(* compensation not necessarily finished if axis stops (new modes available) - 2009-08-13 KSt *)
(*	IF NOT F_AxisHasJob(Axis.NcToPlc.StateDWord) THEN
		/* command aborted, move has been stopped before superposition finished (KSt, 12.01.2004) */
		CommandAborted := TRUE;
		iState := STATE_INITIALIZATION;
	END_IF
*)

STATE_WAITING : (* 2009-10-06 KSt  - state added for axes coupled to actual position (encoder axes or disabled axes) *)
	(* decide if superposition was completed or aborted in case of axes coupled to actual position (encoder axes or disabled axes) *)
	IF NOT F_AxisIsMoving(Axis.NcToPlc.StateDWord) THEN (* 2009-10-06 KSt *)
		(* command aborted, motion ended before superposition was finished because the axis is not moving any longer *)
		CommandAborted := TRUE;
	ELSE
		(* the initial HasJob or Moving state was the same as at end of compensation - assume that superposition completed *)
		Done := TRUE;
	END_IF
	CompensationStarted := FALSE;
	iState := STATE_INITIALIZATION;

ELSE  (* CASE : Unknown program state *)
	Error := TRUE;
	ErrorID := 16#FFFFFFFF;
	iState:= STATE_INITIALIZATION;
END_CASE

ADSbusy := fbAdsReadWrite.BUSY;
IF iState=STATE_INITIALIZATION THEN
	(* reset Busy immediately  when sequence ends *)
	IF Busy THEN
		LastExecutionResult.Done := Done;
		LastExecutionResult.CommandAborted := CommandAborted;
		LastExecutionResult.Error := Error;
		LastExecutionResult.ErrorID := ErrorID;
	END_IF
	Busy := FALSE;
	Active := FALSE;
END_IF
END_FUNCTION_BLOCK

(* POU MC_OverrideFilter, ST *)
FUNCTION_BLOCK MC_OverrideFilter
VAR_INPUT
	(* variables *)
	OverrideValueRaw		: DINT;
	(* parameter *)
	LowerOverrideThreshold	: DINT	:= 0;			(* 0...32767 digits *)
	UpperOverrideThreshold	: DINT	:= 32767;		(* 0...32767 digits *)
	OverrideSteps			: UDINT	:= 200;		(* 200 steps => 0.5 percent *)
	OverrideRecoveryTime	: TIME	:= T#150ms;	(* 150 ms *)
END_VAR
VAR_OUTPUT
	OverrideValueFiltered		: DWORD;			(* 0...1000000 counts *)
	OverridePercentFiltered	: LREAL;				(* 0...100 % *)
	Error					: BOOL;
	ErrorID					: UDINT;
END_VAR
VAR
	bFirstCycle				: BOOL := TRUE;
	bThresholdActive			: BOOL := TRUE;
	InternalOverrideValueRaw	: DINT;
	LastOverrideValueRaw		: DINT := 16#FFFF;
	OverrideRange			: DINT;
END_VAR
{library private}
VAR
	fbTimer					: TON;
END_VAR
(* default value *)
Error	:= FALSE;
ErrorID	:= MC_ERROR_NO_ERROR;

(* check parameter / error handling:   'UpperOverrideThreshold > LowerOverrideThreshold'  AND  'OverrideSteps > 1'  *)
IF( (LowerOverrideThreshold >= UpperOverrideThreshold) OR (OverrideSteps <= 1) )THEN
	OverrideValueFiltered		:= 0;
	OverridePercentFiltered	:= 0.0;
	Error	:= TRUE;
	ErrorID	:= MC_ERROR_PARAMETER_NOT_CORRECT;
	RETURN;
END_IF;

(* first cycle: timer must be elapsed *)
IF ( bFirstCycle ) THEN
	fbTimer( IN:=TRUE, PT:= T#0s );
	bFirstCycle := FALSE;
END_IF;

IF ( OverrideValueRaw >= UpperOverrideThreshold ) THEN
	InternalOverrideValueRaw := UpperOverrideThreshold;
	bThresholdActive := TRUE;
ELSIF ( OverrideValueRaw <= LowerOverrideThreshold ) THEN
	InternalOverrideValueRaw := LowerOverrideThreshold;
	bThresholdActive := TRUE;
ELSE
	InternalOverrideValueRaw := OverrideValueRaw;
	bThresholdActive := FALSE;
END_IF;

fbTimer( IN:=TRUE, PT:= OverrideRecoveryTime );
IF( fbTimer.Q = TRUE OR bThresholdActive )THEN
	OverrideRange := UpperOverrideThreshold - LowerOverrideThreshold;
(*	IF (  bThresholdActive OR ABS( InternalRawOverrideValue - LastRawOverrideValue ) >= (0.5 * OverrideRange / OverrideSteps)  ) THEN *)
	IF (  bThresholdActive OR ABS( InternalOverrideValueRaw - LastOverrideValueRaw ) >= ( OverrideRange / OverrideSteps)  ) THEN
		OverrideValueFiltered := ((InternalOverrideValueRaw - LowerOverrideThreshold) * 1000 / OverrideRange) * 1000;
		OverridePercentFiltered := DWORD_TO_LREAL( OverrideValueFiltered ) * 0.0001;
		LastOverrideValueRaw := InternalOverrideValueRaw;
		fbTimer( IN:=FALSE, PT:= OverrideRecoveryTime );
	END_IF;
END_IF;
END_FUNCTION_BLOCK

(* POU MC_Power, ST *)
FUNCTION_BLOCK MC_Power
(*
	Function block defined by PLCopen Part 1 - Function blocks for motion control

	This Function Block controls the power stage (on or off).
*)
VAR_IN_OUT
	Axis				:	AXIS_REF;	(* B *)
END_VAR
VAR_INPUT
	Enable			:	BOOL;	(* B *)
	Enable_Positive	:	BOOL;	(* E *)
	Enable_Negative	:	BOOL;	(* E *)
	Override			:	LREAL	(* V *) 	:= 100.0; (* in percent - Beckhoff proprietary input *)
	BufferMode		:	MC_BufferMode;	(* E *)
END_VAR
VAR_OUTPUT
	Status			:	BOOL;	(* B *)
	Busy			: 	BOOL;	(* E *)
	Active			: 	BOOL;	(* E *)
	Error			:	BOOL;	(* B *)
	ErrorID			:	UDINT;	(* E *)
END_VAR
{library private}
VAR
	EnableTimeout: TON;
	EnableOffOnDelay: TP;
	iOverride: DINT;
END_VAR
(*EnableTimeout(IN:=Enable, PT:=T#10s);*)	(* timout if axis doesn't get ready after Enable *)
EnableTimeout(IN:=Enable AND NOT Status AND Axis.NcToPlc.CoupleState=0, PT:=T#10s);	(* timout if axis doesn't get ready after Enable - just for single axes - KSt 2010-03-11 *)
EnableOffOnDelay(IN:= NOT Enable );	(* minimum delay between disable end re-Enable -  don't initialize before first enable *)

IF Enable THEN
	Busy := TRUE;
	Status := FALSE;
	ErrorID := 0;
	Error := FALSE;
	EnableOffOnDelay.PT:=T#50ms;	(* initialize not before first enable *)

	(* set override *)
	iOverride := LREAL_TO_UDINT(Override*10000);
	(* double check override with real and integer number because conversion may fail *)
	IF (Override < -1) OR (Override > 101) THEN	(* check real number with tolerance *)
		ErrorID := MC_ERROR_PARAMETER_NOT_CORRECT;
		Error := TRUE;
	ELSIF (iOverride < 0) OR (iOverride > 1000000) THEN	(* check integer number without tolerance *)
		ErrorID := MC_ERROR_PARAMETER_NOT_CORRECT;
		Error := TRUE;
	ELSE
		Axis.PlcToNc.Override := iOverride;
	END_IF;

	(* set enabling flags *)
	Axis.PlcToNc.ControlDWord.0 := Enable;
	Axis.PlcToNc.ControlDWord.1 := Enable_Positive;
	Axis.PlcToNc.ControlDWord.2 := Enable_Negative;

	(* set status bit *)
	(* IF  F_AxisIsReady(StateDWord := Axis.NcToPlc.StateDWord) THEN *) (* Axis ready*) 	(* 2008-12-18 KSt *)
	IF  F_AxisControlLoopClosed(StateDWord := Axis.NcToPlc.StateDWord) THEN (* Axis ready*) 	(* 2008-12-18 KSt *)
		(* status is TRUE if no error and a minimum of EnableOffOnDelay.PT (50 ms) after last recent disable *)
		Status := NOT Error AND NOT EnableOffOnDelay.Q; (* exclusive outputs *)
	ELSIF Axis.Status.ErrorID <> 0 THEN (* 2009-01-29 KSt *)
		Status := FALSE;
		Error := TRUE;
		ErrorID := Axis.Status.ErrorID;
	ELSIF EnableTimeout.Q THEN
		(* timeout after enable *)
		Status := FALSE;
		Error := TRUE;
		ErrorID := MC_ERROR_AXIS_IS_NOT_READY;
	END_IF;

ELSE (* NOT Enable *)
	(* if BufferMode=Buffered wait for current command beeing finished *)
	IF BufferMode = MC_Aborting OR NOT F_AxisHasJob(Axis.NcToPlc.StateDWord) THEN
		Axis.PlcToNc.ControlDWord:= CLEARBIT32(Axis.PlcToNc.ControlDWord,0);
		Axis.PlcToNc.ControlDWord:= CLEARBIT32(Axis.PlcToNc.ControlDWord,1);
		Axis.PlcToNc.ControlDWord:= CLEARBIT32(Axis.PlcToNc.ControlDWord,2);
		(* Override  0 % *)
		Axis.PlcToNc.Override := 0;
		Status := FALSE;
		Busy := FALSE;
		Error := FALSE;			(* reset at falling edge of Execute *)
		ErrorID := 0;
	END_IF
END_IF;

Active:=TRUE;
END_FUNCTION_BLOCK

(* POU MC_PowerStepper, ST *)
FUNCTION_BLOCK MC_PowerStepper
VAR_IN_OUT
	Axis		:	AXIS_REF;
END_VAR
VAR_INPUT
	Enable			:	BOOL;
	Enable_Positive	:	BOOL;
	Enable_Negative	:	BOOL;
	Override			:	LREAL := 100.0; (* in percent *)
	DestallParams	:	ST_PowerStepperStruct;
	KL_Status		:	USINT;
	KL_Status2		:	UINT;
END_VAR
VAR_OUTPUT
	Status			:	BOOL;
	Error			:	BOOL;
	ErrorID			:	UDINT;
	Stalled			:	BOOL;
	StallError			:	BOOL;
END_VAR
VAR
	fbPower			:	MC_Power;
	ErrorCode		:	DWORD;
	fbWriteErrCode	:	ADSWRITE;
	nRefState		:	DWORD;
	fbWriteNonRef	:	ADSWRITE;
	fbReadParams	:	ADSREAD;
	fbWriteInstOvr		:	ADSWRITE;
	bAdsInitDone		:	BOOL;

	bOverTemp		:	BOOL;
	rtOverTemp		:	R_TRIG;
	bUnderVoltage	:	BOOL;
	rtUnderVoltage	:	R_TRIG;
	bOpenLoopA		:	BOOL;
	rtOpenLoopA		:	R_TRIG;
	bOpenLoopB		:	BOOL;
	rtOpenLoopB		:	R_TRIG;
	bOverCurrentA	:	BOOL;
	rtOverCurrentA	:	R_TRIG;
	bOverCurrentB	:	BOOL;
	rtOverCurrentB	:	R_TRIG;
	rtStallError		:	R_TRIG;
	bOldState		:	BOOL;

	bLagFilterInit		: 	BOOL;
	tonLagFilter		:	TON;
	tonNoLagFilter	:	TON;

	wState2			:	WORD;
	nAngle			:	INT;
	nOldAngle		:	INT;
	AngleDiff			:	INT;
	bInErrorState		:	BOOL;

	nParamIdx		:	INT;
	bParamEnabled	:	BOOL;
	fLagLimit			:	LREAL;
	fLagFilter			:	LREAL;
	nTries			:	INT;
	tTimeOut			:	TON;
END_VAR
(*
	Aufruf des Standard-Bausteins
*)
fbPower(
	Enable:=Enable,
	Enable_Positive:=Enable_Positive,
	Enable_Negative:=Enable_Negative,
	Override:=Override,
	Axis:=Axis);

(*
	Ein paar Vorbereitungen ...
*)
wState2:=UINT_TO_WORD(KL_Status2);
bInErrorState:=Axis.NcToPlc.ErrorCode<>0;
nAngle:=SHR(USINT_TO_BYTE(KL_Status),1) AND 7;
AngleDiff:=nAngle-nOldAngle;
nOldAngle:=nAngle;
IF((Axis.NcToPlc.StateDWord AND 16#0000001C)=16#0000001C)THEN		(* Ziel erreicht *)
	nTries:=0;
END_IF
IF((Axis.NcToPlc.StateDWord AND 16#00000080)=16#00000080)THEN		(* Stop *)
	nTries:=0;
END_IF

(* ======================================
	Parameter-Lademaschine
====================================== *)
IF(NOT Enable)THEN
	(*
		Reinitialisieren
	*)
	nParamIdx:=0;
	bParamEnabled:=FALSE;
	fbReadParams(
		NETID:='', PORT:=AMSPORT_R0_NCSAF, IDXGRP:=0, IDXOFFS:=0,
		LEN:=0, DESTADDR:=0,
		READ:=FALSE, TMOUT:=T#5s);
ELSE
	IF(NOT bParamEnabled)THEN
		CASE nParamIdx OF
			0:
				IF(NOT fbReadParams.READ)THEN
					fbReadParams.LEN:=SIZEOF(fLagLimit);
					fbReadParams.DESTADDR:=ADR(fLagLimit);
					fbReadParams.IDXGRP:=16#00004000+Axis.NcToPlc.AxisId;
					fbReadParams.IDXOFFS:=16#00020012;
					fbReadParams.READ:=TRUE;
				ELSIF(NOT fbReadParams.BUSY)THEN
					IF(fbReadParams.ERR)THEN
						fLagLimit:=5.0;
					END_IF
					fbReadParams.READ:=FALSE;
					nParamIdx:=nParamIdx+1;
				END_IF
				fbReadParams(NETID:='', PORT:=AMSPORT_R0_NCSAF, TMOUT:=T#5s);
			1:
				IF(NOT fbReadParams.READ)THEN
					fbReadParams.LEN:=SIZEOF(fLagFilter);
					fbReadParams.DESTADDR:=ADR(fLagFilter);
					fbReadParams.IDXGRP:=16#00004000+Axis.NcToPlc.AxisId;
					fbReadParams.IDXOFFS:=16#00020013;
					fbReadParams.READ:=TRUE;
				ELSIF(NOT fbReadParams.BUSY)THEN
					IF(fbReadParams.ERR)THEN
						fLagFilter:=0.1;
					END_IF
					fbReadParams.READ:=FALSE;
					nParamIdx:=nParamIdx+1;
					tonLagFilter(IN:=FALSE, PT:=T#10ms);
					tonNoLagFilter(IN:=NOT tonLagFilter.IN, PT:=T#10ms);
				END_IF
				fbReadParams(NETID:='', PORT:=AMSPORT_R0_NCSAF, TMOUT:=T#5s);
			ELSE
				bParamEnabled:=TRUE;
		END_CASE
	END_IF
END_IF

IF(fbPower.Error)THEN
	ErrorID := fbPower.ErrorID;
	Error := TRUE;
	Status := bAdsInitDone := FALSE;
ELSIF(NOT Enable)THEN
	ErrorID := 0;
	Error := Status := bAdsInitDone := FALSE;
ELSE
	(*
		Sicherstellen, dass die ADS-FBs initialisiert sind
	*)
	IF(NOT bAdsInitDone)THEN
		bAdsInitDone := TRUE;
		fbWriteNonRef(
			WRITE:=FALSE,
			NETID:='',
			PORT:=AMSPORT_R0_NCSAF,
			IDXGRP:=16#00004200+Axis.NcToPlc.AxisId,
			IDXOFFS:=16#0000001B,
			LEN:=SIZEOF(nRefState),
			SRCADDR:=ADR(nRefState),
			TMOUT:=T#5s,
			);
		fbWriteInstOvr(
			WRITE:=FALSE,
			NETID:='',
			PORT:=AMSPORT_R0_NCSAF,
			IDXGRP:=16#00004200+Axis.NcToPlc.AxisId,
			IDXOFFS:=16#00000029,
			LEN:=0,
			SRCADDR:=0,
			TMOUT:=T#5s,
			);
		fbWriteErrCode(
			WRITE:=FALSE,
			NETID:='',
			PORT:=AMSPORT_R0_NCSAF,
			IDXGRP:=16#00004200+Axis.NcToPlc.AxisId,
			IDXOFFS:=16#00000019,
			LEN:=SIZEOF(ErrorCode),
			SRCADDR:=ADR(ErrorCode),
			TMOUT:=T#5s,
			);
	END_IF

	(*
		Zentrales Versenden für Kommandos zur instantanen Override-Änderung
		Dies muss vor der Stelle des Test liegen, damit der Override-Wert im Mapping sicher angekommen ist,
		wenn dieses Kommando per ADS eintrifft.
	*)
	fbWriteInstOvr(
		NETID:='',
		PORT:=AMSPORT_R0_NCSAF,
		IDXGRP:=16#00004200+Axis.NcToPlc.AxisId,
		IDXOFFS:=16#00000029,
		LEN:=0,
		SRCADDR:=0,
		TMOUT:=T#5s,
		);
	IF(NOT fbWriteInstOvr.BUSY)THEN
		fbWriteInstOvr.WRITE:=FALSE;
	END_IF

	bLagFilterInit:=bLagFilterInit OR tonLagFilter.Q;

	IF(DestallParams.DestallEnable)THEN
		(*
			Stall Detection
		*)
		bOldState:=Stalled;
		CASE DestallParams.DestallDetectMode OF
			PwStDetectMode_Encoderless:
				Stalled:=ABS(AngleDiff)>=4;
			PwStDetectMode_Lagging:
				IF(bParamEnabled)THEN
					IF(fLagFilter<=0.001)THEN
						tonLagFilter(IN:=FALSE, PT:=T#10ms);
						tonNoLagFilter(IN:=NOT tonLagFilter.IN, PT:=T#10ms);
						Stalled:=ABS(Axis.NcToPlc.PosDiff)>=fLagLimit;
					ELSE
						tonLagFilter(IN:=(ABS(Axis.NcToPlc.PosDiff)>=fLagLimit), PT:=LREAL_TO_TIME(fLagFilter*1000.0));
						tonNoLagFilter(IN:=NOT tonLagFilter.IN, PT:=LREAL_TO_TIME(fLagFilter*1000.0));
						Stalled:=tonLagFilter.Q;
					END_IF
				ELSE
					tonLagFilter(IN:=FALSE, PT:=T#10ms);
					tonNoLagFilter(IN:=NOT tonLagFilter.IN, PT:=T#10ms);
					Stalled:=FALSE;
				END_IF
			ELSE
				Stalled:=FALSE;
		END_CASE
		IF(NOT bOldState AND Stalled)THEN
			nTries:=nTries+1;
		END_IF
		(*
			Stall Handling
		*)
		StallError:=StallError AND (bInErrorState  OR fbWriteErrCode.WRITE);
		bOldState:=StallError;
		CASE DestallParams.DestallMode OF
			PwStMode_None:
				StallError:=FALSE;
				tTimeOut(IN:=FALSE, PT:=T#10ms);
			PwStMode_SetError:
				StallError:=StallError OR Stalled;
				tTimeOut(IN:=FALSE, PT:=T#10ms);
			PwStMode_SetErrNonRef:
				StallError:=StallError OR Stalled;
				IF(Stalled AND ((Axis.NcToPlc.StateDWord AND 16#00000002)<>0) )THEN
					nRefState:=0;
					fbWriteNonRef.WRITE:=TRUE;
				END_IF
				tTimeOut(IN:=FALSE, PT:=T#10ms);
			PwStMode_UseOverride:
				IF(Stalled OR (bLagFilterInit AND NOT tonNoLagFilter.Q))THEN	(* HKP *)
					Axis.PlcToNc.Override := 0;
					fbWriteInstOvr.WRITE:=TRUE;
				END_IF
				tTimeOut(IN:=Stalled, PT:=MAX(DestallParams.Timeout, T#10ms));
				StallError:=StallError OR tTimeOut.Q;
				IF(nTries>DestallParams.Retries)THEN
					StallError:=TRUE;
				END_IF
		END_CASE

		IF(StallError AND NOT bOldState)THEN
			ADSLOGDINT((ADSLOG_MSGTYPE_ERROR OR ADSLOG_MSGTYPE_LOG), 'MC_PowerStepper (AxisID: %d) reporting error 0x4636 (stall error) !', Axis.NcToPlc.AxisId);
		END_IF
		rtStallError(CLK:=StallError AND NOT bInErrorState AND NOT fbWriteErrCode.WRITE);
		IF(rtStallError.Q)THEN
			ErrorCode:=16#00004636;
			fbWriteErrCode.WRITE:=TRUE;
		END_IF

	END_IF

	Status:=TRUE;
	IF(DestallParams.StatusMonEnable)THEN
		(*
			State Monitoring
		*)
		bOldState:=bOverTemp;
		bOverTemp:=(wState2 AND 2#0000000100000000)<>0;
		Status:=Status AND NOT bOverTemp;
		IF(bOverTemp AND NOT bOldState)THEN
			ADSLOGDINT((ADSLOG_MSGTYPE_ERROR OR ADSLOG_MSGTYPE_LOG), 'MC_PowerStepper (AxisID: %d) reporting error 0x4630 (overtemperature, KL terminal) !', Axis.NcToPlc.AxisId);
		END_IF
		rtOverTemp(CLK:=bOverTemp AND NOT bInErrorState AND NOT fbWriteErrCode.WRITE);
		IF(rtOverTemp.Q)THEN
			ErrorCode:=16#00004630;
			fbWriteErrCode.WRITE:=TRUE;
		END_IF
		bOverTemp:=bOverTemp AND (bInErrorState  OR fbWriteErrCode.WRITE);
		bOldState:=bUnderVoltage;
		bUnderVoltage:=(wState2 AND 2#0000001000000000)<>0;
		Status:=Status AND NOT bUnderVoltage;
		IF(bUnderVoltage AND NOT bOldState)THEN
						ADSLOGDINT((ADSLOG_MSGTYPE_ERROR OR ADSLOG_MSGTYPE_LOG), 'MC_PowerStepper (AxisID: %d) reporting error 0x4631 (bad supply voltage, KL terminal) !', Axis.NcToPlc.AxisId);
		END_IF
		rtUnderVoltage(CLK:=bUnderVoltage AND NOT bInErrorState AND NOT fbWriteErrCode.WRITE);
		IF(rtUnderVoltage.Q)THEN
			ErrorCode:=16#00004631;
			fbWriteErrCode.WRITE:=TRUE;
		END_IF
		bUnderVoltage:=bUnderVoltage AND (bInErrorState  OR fbWriteErrCode.WRITE);
		bOldState:=bOpenLoopA;
		bOpenLoopA:=(wState2 AND 2#0000010000000000)<>0;
		Status:=Status AND NOT bOpenLoopA;
		IF(bOpenLoopA AND NOT bOldState)THEN
			ADSLOGDINT((ADSLOG_MSGTYPE_ERROR OR ADSLOG_MSGTYPE_LOG), 'MC_PowerStepper (AxisID: %d) reporting error 0x4632 (open loop, phase A) !', Axis.NcToPlc.AxisId);
		END_IF
		rtOpenLoopA(CLK:=bOpenLoopA AND NOT bInErrorState AND NOT fbWriteErrCode.WRITE);
		IF(rtOpenLoopA.Q)THEN
			ErrorCode:=16#00004632;
			fbWriteErrCode.WRITE:=TRUE;
		END_IF
		bOpenLoopA:=bOpenLoopA AND (bInErrorState  OR fbWriteErrCode.WRITE);
		bOldState:=bOpenLoopB;
		bOpenLoopB:=(wState2 AND 2#0000100000000000)<>0;
		Status:=Status AND NOT bOpenLoopB;
		IF(bOpenLoopB AND NOT bOldState)THEN
			ADSLOGDINT((ADSLOG_MSGTYPE_ERROR OR ADSLOG_MSGTYPE_LOG), 'MC_PowerStepper (AxisID: %d) reporting error 0x4633 (open loop, phase B) !', Axis.NcToPlc.AxisId);
		END_IF
		rtOpenLoopB(CLK:=bOpenLoopB AND NOT bInErrorState AND NOT fbWriteErrCode.WRITE);
		IF(rtOpenLoopB.Q)THEN
			ErrorCode:=16#00004633;
			fbWriteErrCode.WRITE:=TRUE;
		END_IF
		bOpenLoopB:=bOpenLoopB AND (bInErrorState  OR fbWriteErrCode.WRITE);
		bOldState:=bOverCurrentA;
		bOverCurrentA:=(wState2 AND 2#0001000000000000)<>0;
		Status:=Status AND NOT bOverCurrentA;
		IF(bOverCurrentA AND NOT bOldState)THEN
			ADSLOGDINT((ADSLOG_MSGTYPE_ERROR OR ADSLOG_MSGTYPE_LOG), 'MC_PowerStepper (AxisID: %d) reporting error 0x4634 (overcurrent, phase A) !', Axis.NcToPlc.AxisId);
		END_IF
		rtOverCurrentA(CLK:=bOverCurrentA AND NOT bInErrorState AND NOT fbWriteErrCode.WRITE);
		IF(rtOverCurrentA.Q)THEN
			ErrorCode:=16#00004634;
			fbWriteErrCode.WRITE:=TRUE;
		END_IF
		bOverCurrentA:=bOverCurrentA AND (bInErrorState  OR fbWriteErrCode.WRITE);
		bOldState:=bOverCurrentB;
		bOverCurrentB:=(wState2 AND 2#0010000000000000)<>0;
		Status:=Status AND NOT bOverCurrentB;
		IF(bOverCurrentB AND NOT bOldState)THEN
			ADSLOGDINT((ADSLOG_MSGTYPE_ERROR OR ADSLOG_MSGTYPE_LOG), 'MC_PowerStepper (AxisID: %d) reporting error 0x4635 (overcurrent, phase B) !', Axis.NcToPlc.AxisId);
		END_IF
		rtOverCurrentB(CLK:=bOverCurrentB AND NOT bInErrorState AND NOT fbWriteErrCode.WRITE);
		IF(rtOverCurrentB.Q)THEN
			ErrorCode:=16#00004635;
			fbWriteErrCode.WRITE:=TRUE;
		END_IF
		bOverCurrentB:=bOverCurrentB AND (bInErrorState  OR fbWriteErrCode.WRITE);
	END_IF

	(*
		Zentrale Versendung von Achs-ErrorCodes
	*)
	fbWriteErrCode(
		NETID:='',
		PORT:=AMSPORT_R0_NCSAF,
		IDXGRP:=16#00004200+Axis.NcToPlc.AxisId,
		IDXOFFS:=16#00000019,
		LEN:=SIZEOF(ErrorCode),
		SRCADDR:=ADR(ErrorCode),
		TMOUT:=T#5s,
		);
	IF(bInErrorState)THEN
		fbWriteErrCode.WRITE:=FALSE;
	END_IF

	(*
		Zentrale Versendung von Referenz-Resets
	*)
	fbWriteNonRef(
		NETID:='',
		PORT:=AMSPORT_R0_NCSAF,
		IDXGRP:=16#00004200+Axis.NcToPlc.AxisId,
		IDXOFFS:=16#0000001B,
		LEN:=SIZEOF(nRefState),
		SRCADDR:=ADR(nRefState),
		TMOUT:=T#5s,
		);
	IF(NOT fbWriteNonRef.BUSY)THEN
		fbWriteNonRef.WRITE:=FALSE;
	END_IF

END_IF
END_FUNCTION_BLOCK

(* POU MC_ReadActualPosition, ST *)
FUNCTION_BLOCK MC_ReadActualPosition
(*	This Function Block returns the actual position. *)
VAR_IN_OUT
	Axis			:	AXIS_REF;	(* B *)
END_VAR
VAR_INPUT
	Enable		:	BOOL;		(* B *)
END_VAR
VAR_OUTPUT
	Valid		:	BOOL;		(* B *)
	Busy		:	BOOL;		(* E *)
	Error		:	BOOL;		(* B *)
	ErrorID		:	UDINT;		(* E *)
	Position		:	LREAL;		(* B *)
END_VAR
VAR
END_VAR
Error := FALSE;
ErrorID := 0;
IF Enable THEN
	Busy := TRUE;
	Position := Axis.NcToPlc.ActPos;
	Valid := TRUE;
ELSE
	Busy := FALSE;
	Position := 0.0;
	Valid := FALSE;
END_IF;
END_FUNCTION_BLOCK

(* POU MC_ReadActualVelocity, ST *)
FUNCTION_BLOCK MC_ReadActualVelocity
(*
	This Function Block returns the value of the actual velocity as long as Enable is 
	set. Valid is true when the data-output ActualVelocity is valid. If Enable is Reset, the 
	data loses its validity, and Valid is also reset, no matter if new data is available.
*)
VAR_IN_OUT
	Axis			:	AXIS_REF;	(* B *)
END_VAR
VAR_INPUT
	Enable 		: 	BOOL;	(* B *)
END_VAR
VAR_OUTPUT
	Valid 		: 	BOOL;	(* B *)
	Busy 		: 	BOOL;	(* E *)
	Error 		: 	BOOL;	(* B *)
	ErrorID 		: 	UDINT;	(* E *)
	ActualVelocity : 	LREAL;	(* B *)
END_VAR
VAR
END_VAR
Error := FALSE;
ErrorID := 0;
IF Enable THEN
	Busy := TRUE;
	Valid := TRUE;
	ActualVelocity := Axis.NcToPlc.ActVelo;
ELSE
	Busy := FALSE;
	Valid := FALSE;
	ActualVelocity := 0;
END_IF
END_FUNCTION_BLOCK

(* POU MC_ReadAxisComponents, ST *)
FUNCTION_BLOCK  MC_ReadAxisComponents
VAR_IN_OUT
	AxisComponents 	: 	ST_AxisComponents;
	Axis				:	AXIS_REF;
END_VAR
VAR_INPUT
	Execute: BOOL;
END_VAR
VAR_OUTPUT
	Done : BOOL;
	Busy: BOOL;
	Error : BOOL;
	ErrorID : UDINT;
END_VAR
VAR
	TriggerExecute: R_TRIG;
	state: _E_TcMC_STATES := STATE_INITIALIZATION;
	fbAdsRead		: 	ADSREAD;
END_VAR
TriggerExecute(CLK:=Execute);

CASE state OF
	STATE_INITIALIZATION:
		IF NOT Execute THEN
			Done := FALSE;
			Error := FALSE;	(* reset at falling edge of Execute *)
			ErrorID := 0;
		END_IF
		IF TriggerExecute.Q THEN
			Done := FALSE;
			Busy := TRUE;
			Error := FALSE;
			ErrorID := 0;
			fbAdsRead(READ:=FALSE);
		END_IF
		IF Busy THEN
			fbAdsRead(
				NETID:= TcMcGlobal.NCNETID_TCMC,
				PORT:= TcMcGlobal.NCPORT_TCMC,
				IDXGRP:=TcMcGlobal.Axis.Parameter.IDXGRP+Axis.NcToPlc.AxisId,
				IDXOFFS:= 16#5A,
				LEN:= SIZEOF(AxisComponents),
				DESTADDR:= ADR(AxisComponents),
				READ:= TRUE,
				TMOUT:= TcMcGlobal.tADSTimeOut );
			IF NOT fbAdsRead.BUSY THEN
				Error := fbAdsRead.ERR;
				ErrorID := fbAdsRead.ERRID;
				Done := NOT Error;
				Busy := FALSE;
			END_IF
		END_IF
END_CASE
END_FUNCTION_BLOCK

(* POU MC_ReadAxisError, ST *)
FUNCTION_BLOCK MC_ReadAxisError
(*	This Function Block describes general axis errors not relating to the Function Blocks. *)
VAR_IN_OUT
	Axis				:	AXIS_REF;	(* B *)
END_VAR
VAR_INPUT
	Enable			:	BOOL;		(* B *)
END_VAR
VAR_OUTPUT
	Valid			:	BOOL;		(* B *)
	Busy			:	BOOL;		(* E *)
	Error			:	BOOL;		(* B *)
	ErrorID			:	DWORD;	(* B *)
	AxisErrorID		:	DWORD;	(* B *)
END_VAR
VAR
END_VAR
IF Enable THEN
	Busy		 := TRUE;
	Valid 		:=  TRUE;
	ErrorID 		:= 0;
	AxisErrorID 	:= Axis.NcToPlc.ErrorCode;
	Error		:= ErrorID <> 0;
ELSE
	Busy 		:= FALSE;
	Valid 		:= FALSE;
	Error 		:= FALSE;	(* reset at falling edge of Execute *)
	ErrorID 		:= 0;
	AxisErrorID 	:= 0;
END_IF;
END_FUNCTION_BLOCK

(* POU MC_ReadBoolParameter, ST *)
FUNCTION_BLOCK MC_ReadBoolParameter
(*	This Function Block returns the value of a vendor specific boolean parameter.*)
VAR_IN_OUT
	Axis					:	AXIS_REF;	(* B *)
END_VAR
VAR_INPUT
	Enable				:	BOOL;		(* B *)
	ParameterNumber		:	INT;			(* B *)
	ReadMode			:	E_ReadMode(* V *)	:= ReadMode_Once;	 (* Beckhoff proprietary input *)
END_VAR
VAR_OUTPUT
	Valid				:	BOOL;	(* B *)
	Busy				: 	BOOL;	(* E *)
	Error				:	BOOL;	(* B *)
	ErrorID				:	UDINT;	(* E *)
	Value				:	BOOL;	(* B *)
END_VAR
VAR
	ADSbusy: BOOL;
	fbReadWriteParameter: 	_FB_ReadWriteParameter;
END_VAR
{library private}
VAR
	nParatype 			: 	_E_ParameterType;
	dwValue 				: 	DWORD;
	lrValue				: 	LREAL;
	bStarted				:	BOOL;
	fbTrigger 			: 	R_TRIG;
END_VAR
IF NOT Enable THEN
	Valid := FALSE;
	Error := FALSE;			(* reset at falling edge of Execute *)
	ErrorID := 0;
END_IF
IF ReadMode = ReadMode_Once THEN
	fbTrigger(CLK:= Enable);
	IF fbTrigger.Q AND NOT bStarted THEN
		bStarted := TRUE;
		Valid := FALSE;
		Error := FALSE;
		ErrorID := MC_ERROR_NO_ERROR;
	END_IF;
ELSE
	IF Enable AND NOT bStarted THEN
		bStarted := TRUE;
		Valid := FALSE;
		Error := FALSE;
		ErrorID := MC_ERROR_NO_ERROR;
	END_IF;
END_IF;
(* *)
IF bStarted THEN
	nParatype := PARAMETERTYPE_BOOL;
	fbReadWriteParameter(Enable:= TRUE, ParameterNumber:= ParameterNumber, Mode:= READWRITEPARAMETERMODE_READ,
						ParameterType:=nParatype, Axis:= Axis, ValueLreal:= lrValue, ValueDword := dwValue, ValueBool := Value);
	IF fbReadWriteParameter.Done THEN
		bStarted := FALSE;
		Valid := TRUE;
		fbReadWriteParameter(Enable:= FALSE, ParameterNumber:= ParameterNumber, Mode:= READWRITEPARAMETERMODE_READ,
						ParameterType:= nParatype , Axis:= Axis, ValueLreal:= lrValue, ValueDword := dwValue, ValueBool := Value);
	END_IF;
	IF fbReadWriteParameter.Error THEN
		bStarted := FALSE;
		Valid := FALSE;
		Error := TRUE;
		ErrorID := fbReadWriteParameter.ErrorID;
		fbReadWriteParameter(Enable:= FALSE, ParameterNumber:= ParameterNumber, Mode:= READWRITEPARAMETERMODE_READ,
						ParameterType:= nParatype , Axis:= Axis, ValueLreal:= lrValue, ValueDword := dwValue, ValueBool := Value);
	END_IF;
END_IF;

ADSbusy := fbReadWriteParameter.ADSbusy;
Busy := (Enable AND ReadMode<>ReadMode_Once) OR bStarted;
END_FUNCTION_BLOCK

(* POU MC_ReadDriveAddress, ST *)
FUNCTION_BLOCK MC_ReadDriveAddress
(*	This Function Block returns the value of a vendor specific parameter *)
VAR_IN_OUT
	Axis				: AXIS_REF;	(* B *)
END_VAR
VAR_INPUT
	Execute			: BOOL;
END_VAR
VAR_OUTPUT
	Done 			: BOOL;
	Busy			: BOOL;
	Error			: BOOL;
	ErrorID			: UDINT;
	DriveAddress 	: ST_DriveAddress;
END_VAR
VAR
	state			: 	_E_TcMC_STATES := STATE_INITIALIZATION;
	TriggerExecute: R_TRIG;
	fbAdsRead: ADSREAD;
	readBuffer			: ARRAY[0..9] OF BYTE;
	i: INT;
END_VAR
TriggerExecute(CLK:=Execute);

CASE state OF
	STATE_INITIALIZATION:
		IF NOT Execute THEN
			Done := FALSE;
			Error := FALSE;	(* reset at falling edge of Execute *)
			ErrorID := 0;
		END_IF
		IF TriggerExecute.Q THEN
			Done := FALSE;
			Busy := TRUE;
			Error := FALSE;
			ErrorID := 0;
			fbAdsRead(READ:=FALSE);
			fbAdsRead(
				NETID:= TcMcGlobal.NCNETID_TCMC,
				PORT:= TcMcGlobal.NCPORT_TCMC,
				IDXGRP:=TcMcGlobal.Axis.Parameter.IDXGRP+Axis.NcToPlc.AxisId,
				IDXOFFS:= TcMcGlobal.Axis.Parameter.IDXOFFS.HWAMSADDR,
				LEN:= SIZEOF(readBuffer),
				DESTADDR:= ADR(readBuffer),
				READ:= TRUE,
				TMOUT:= TcMcGlobal.tADSTimeOut );
			state := STATE_ORDER;
		END_IF

STATE_ORDER:  (* wait until command is accepted *)
		fbAdsRead();
		IF NOT fbAdsRead.BUSY THEN
			Error := fbAdsRead.ERR;
			ErrorID := fbAdsRead.ERRID;
			IF NOT Error THEN
				FOR i := 0 TO 5 DO
					DriveAddress.NetIdBytes[i] := readBuffer[i];
				END_FOR
				DriveAddress.NetID := F_CreateAmsNetId( DriveAddress.NetIdBytes );
				DriveAddress.SlaveAddress := readBuffer[6] + 256* readBuffer[7];
				DriveAddress.Channel := readBuffer[8];
			END_IF
			Done := NOT Error;
			Busy := FALSE;
			fbAdsRead(READ:=FALSE);
			state := STATE_INITIALIZATION;  (* wait until command is accepted *)
		END_IF
END_CASE
END_FUNCTION_BLOCK

(* POU MC_ReadParameter, ST *)
FUNCTION_BLOCK MC_ReadParameter
(*	This Function Block returns the value of a vendor specific parameter *)
VAR_IN_OUT
	Axis				:	AXIS_REF;	(* B *)
END_VAR
VAR_INPUT
	Enable			:	BOOL;		(* B *)
	ParameterNumber	:	INT;			(* B *)
	ReadMode		:	E_ReadMode(* V *) := ReadMode_Once;	 (* Beckhoff proprietary input *)
END_VAR
VAR_OUTPUT
	Valid			:	BOOL;		(* B *)
	Busy			: 	BOOL;		(* E *)
	Error			:	BOOL;		(* B *)
	ErrorID			:	UDINT;		(* E *)
	Value			:	LREAL;		(* B *)
END_VAR
VAR
	ADSbusy		: 	BOOL;
	fbReadWriteParameter: 	_FB_ReadWriteParameter;
END_VAR
{library private}
VAR
	nParatype 		: 	_E_ParameterType;
	dwValue 			: 	DWORD;
	bValue 			: 	BOOL;
	bStarted			:	BOOL;
	fbTrigger		 	: 	R_TRIG;
END_VAR
(* ====================================================================== *)
(* *)
(* ====================================================================== *)
IF NOT Enable THEN
	Valid := FALSE;
	Error := FALSE;			(* reset at falling edge of Execute - just ErrorID will be kept til next rising edge *)
	ErrorID := 0;
END_IF
IF ReadMode = ReadMode_Once THEN
	fbTrigger(CLK:= Enable);
	IF fbTrigger.Q AND NOT bStarted THEN
		bStarted := TRUE;
		Valid := FALSE;
		Error := FALSE;
		ErrorID := MC_ERROR_NO_ERROR;
	END_IF;
ELSE
	IF Enable AND NOT bStarted THEN
		bStarted := TRUE;
		Valid := FALSE;
		Error := FALSE;
		ErrorID := MC_ERROR_NO_ERROR;
	END_IF;
	IF NOT Enable AND NOT bStarted THEN
		Valid := FALSE;
		Error := FALSE;
		ErrorID := MC_ERROR_NO_ERROR;
	END_IF;
END_IF;

IF bStarted THEN
	nParatype := PARAMETERTYPE_LREAL;
	fbReadWriteParameter(Enable:= TRUE, ParameterNumber:= ParameterNumber, Mode:= READWRITEPARAMETERMODE_READ,
						ParameterType:=nParatype, Axis:= Axis, ValueLreal:= Value, ValueDword := dwValue, ValueBool := bValue);
	IF fbReadWriteParameter.Done THEN
		bStarted := FALSE;
		Valid := TRUE;
		fbReadWriteParameter(Enable:= FALSE, ParameterNumber:= ParameterNumber, Mode:= READWRITEPARAMETERMODE_READ,
						ParameterType:= nParatype , Axis:= Axis, ValueLreal:= Value, ValueDword := dwValue, ValueBool := bValue);
	END_IF;
	IF fbReadWriteParameter.Error THEN
		bStarted := FALSE;
		Valid := FALSE;
		Error := TRUE;
		ErrorID := fbReadWriteParameter.ErrorID;
		fbReadWriteParameter(Enable:= FALSE, ParameterNumber:= ParameterNumber, Mode:= READWRITEPARAMETERMODE_READ,
						ParameterType:= nParatype , Axis:= Axis, ValueLreal:= Value, ValueDword := dwValue, ValueBool := bValue);
	END_IF;
END_IF;

ADSbusy := fbReadWriteParameter.ADSbusy;
Busy := (Enable AND ReadMode<>ReadMode_Once) OR bStarted;
END_FUNCTION_BLOCK

(* POU MC_ReadParameterSet, ST *)
FUNCTION_BLOCK  MC_ReadParameterSet
(*	This Function Block returns the complete set of axis parameters *)
VAR_IN_OUT
	Parameter 	: 	ST_AxisParameterSet;
	Axis			:	AXIS_REF;
END_VAR
VAR_INPUT
	Execute		: 	BOOL;
END_VAR
VAR_OUTPUT
	Done 		: 	BOOL;
	Busy		: 	BOOL;
	Error 		: 	BOOL;
	ErrorID 		: 	UDINT;
END_VAR
VAR
	TriggerExecute: R_TRIG;
	state: _E_TcMC_STATES := STATE_INITIALIZATION;
	fbAdsRead		: 	ADSREAD;
END_VAR
TriggerExecute(CLK:=Execute);

CASE state OF
	STATE_INITIALIZATION:
		IF NOT Execute THEN
			Done := FALSE;
			Error := FALSE;	(* reset at falling edge of Execute *)
			ErrorID := 0;
		END_IF
		IF TriggerExecute.Q THEN
			Done := FALSE;
			Busy := TRUE;
			Error := FALSE;
			ErrorID := 0;
			fbAdsRead(READ:=FALSE);
		END_IF
		IF Busy THEN
			fbAdsRead(
				NETID:= TcMcGlobal.NCNETID_TCMC,
				PORT:= TcMcGlobal.NCPORT_TCMC,
				IDXGRP:=TcMcGlobal.Axis.Parameter.IDXGRP+Axis.NcToPlc.AxisId,
				IDXOFFS:= (* 16#00 + *) Axis.NcToPlc.ControlLoopIndex * 16#00100000,
				LEN:= SIZEOF(Parameter),
				DESTADDR:= ADR(Parameter),
				READ:= TRUE,
				TMOUT:= TcMcGlobal.tADSTimeOut );
			IF NOT fbAdsRead.BUSY THEN
				Error := fbAdsRead.ERR;
				ErrorID := fbAdsRead.ERRID;
				Done := NOT Error;
				Busy := FALSE;
			END_IF
		END_IF
END_CASE
END_FUNCTION_BLOCK

(* POU MC_ReadStatus, ST *)
FUNCTION_BLOCK MC_ReadStatus
(*	This Function Block returns in detail the status of the axis with respect to the motion currently in progress *)
VAR_IN_OUT
	Axis				:	AXIS_REF;	(* B *)
END_VAR
VAR_INPUT
	Enable			:	BOOL;	(* B *)
END_VAR
VAR_OUTPUT
	Valid			:	BOOL;	(* B *)
	Busy			: 	BOOL;	(* E *)
	Error			:	BOOL;	(* B *)
	ErrorID			:	UDINT;	(* E *)
	(* motion control statemachine states: *)
	ErrorStop		:	BOOL;	(* B *)
	Disabled			:	BOOL;	(* B *)
	Stopping			:	BOOL;	(* B *)
	StandStill		:	BOOL;	(* B *)
	DiscreteMotion	:	BOOL;	(* B *)
	ContinuousMotion	:	BOOL;	(* B *)
	SynchronizedMotion:	BOOL;	(* E *)
	Homing			:	BOOL;	(* E *)
	(* additional status *)
	ConstantVelocity	:	BOOL;	(* E *)
	Accelerating		:	BOOL;	(* E *)
	Decelerating		:	BOOL;	(* E *)
	(* status data structure *)
	Status			: 	ST_AxisStatus;	(* V *)
END_VAR
VAR
END_VAR
IF Enable THEN
	Busy := TRUE;
	Axis.ReadStatus;
	Status := Axis.Status;

	Error			:= 	Status.Error;
	ErrorID			:= 	Status.ErrorID;

	(* motion control statemachine states: *)
	ErrorStop		:= 	Status.ErrorStop;
	Disabled			:= 	Status.Disabled;
	Stopping			:= 	Status.Stopping;
	StandStill		:= 	Status.StandStill;
	DiscreteMotion	:= 	Status.DiscreteMotion;
	ContinuousMotion	:= 	Status.ContinuousMotion;
	SynchronizedMotion:= 	Status.SynchronizedMotion;
	Homing			:= 	Status.Homing;

	(* additional status *)
	ConstantVelocity	:= 	Status.ConstantVelocity;
	Accelerating		:= 	Status.Accelerating;
	Decelerating		:= 	Status.Decelerating;

	Valid := TRUE;
ELSE
	Busy := FALSE;
	Valid := FALSE;
	Error := FALSE;	(* reset at falling edge of Execute *)
	ErrorID := 0;
END_IF
END_FUNCTION_BLOCK

(* POU MC_Reset, ST *)
FUNCTION_BLOCK MC_Reset
(*
	Function block defined by PLCopen Part 1 - Function blocks for motion control

	This Function Block makes the transition from the state ErrorStop to StandStill
	by resetting all internal axis-related errors. It does not affect the output of the 
	FB instances.
*)
VAR_IN_OUT
	Axis				:	AXIS_REF;	(* B *)
END_VAR
VAR_INPUT
	Execute			:	BOOL;		(* B *)
END_VAR
VAR_OUTPUT
	Done			:	BOOL;		(* B *)
	Busy			:	BOOL;		(* E *)
	Error			:	BOOL;		(* B *)
	ErrorID			:	UDINT;		(* B *)
END_VAR
VAR
	ADSbusy		: 	BOOL;
	iState			:	_E_TcMC_STATES := STATE_INITIALIZATION;
	LastExecutionResult: 	_ST_FunctionBlockResults;
END_VAR
{library private}
VAR
	fbAdsWrite		:	ADSWRITE;
	fbOnTrigger		:	R_TRIG;
END_VAR
fbOnTrigger(CLK:= Execute);

CASE iState OF
	STATE_INITIALIZATION: (* initial iState *)
		Busy := FALSE;
		IF NOT Execute THEN
			Done := FALSE;
			Error := FALSE;			(* reset at falling edge of Execute *)
			ErrorID := 0;
		END_IF
		IF fbOnTrigger.Q THEN
			Busy := TRUE;
			Done:= FALSE;
			Error := FALSE;
			ErrorID := 0;
			fbAdsWrite(WRITE:=FALSE);

			fbAdsWrite(	NETID:= TcMcGlobal.NCNETID_TCMC,
						PORT:= TcMcGlobal.NCPORT_TCMC,
						IDXGRP:=TcMcGlobal.Axis.Functions.IDXGRP+Axis.NcToPlc.AxisId,
						IDXOFFS:= TcMcGlobal.Axis.Functions.IDXOFFS.RESET,
						LEN:= 0,
						SRCADDR:= 0 ,
						WRITE:=TRUE ,
						TMOUT:= TcMcGlobal.tADSTimeOut);
			iState := STATE_ORDER;
		END_IF;

	STATE_ORDER:
		fbAdsWrite();
		 IF NOT fbAdsWrite.Busy THEN
			IF fbAdsWrite.Err THEN
				ErrorID := fbAdsWrite.ErrId;
				Error := TRUE;
			ELSE
				ErrorID := Axis.NcToPlc.ErrorCode;
				Error := ErrorID <> 0;
				Done := NOT Error;
			END_IF;
			fbAdsWrite(WRITE:=FALSE);
			Axis.PlcToNc.PlcCycleControl.1 := 0; (* KSt - 2009-08 - reset exceeded flag for external set point generator *)
			iState := STATE_INITIALIZATION;
		END_IF

	ELSE  (* CASE : Unknown program state *)
		Error := TRUE;
		ErrorID := 16#FFFFFFFF;
		iState:= STATE_INITIALIZATION;
END_CASE;

ADSbusy := fbAdsWrite.BUSY;

IF iState=STATE_INITIALIZATION THEN
	(* reset Busy immediately  when sequence ends *)
	IF Busy THEN
		LastExecutionResult.Done := Done;
		LastExecutionResult.Error := Error;
		LastExecutionResult.ErrorID := ErrorID;
	END_IF
	Busy := FALSE;
END_IF
END_FUNCTION_BLOCK

(* POU MC_SetEncoderScalingFactor, ST *)
FUNCTION_BLOCK MC_SetEncoderScalingFactor
(*
	This function can change the encoder scaling factor in stand-still or on the fly.
*)
VAR_IN_OUT
	Axis			:	AXIS_REF;	(* B *)	(* Identifies the axis to work upon *)
END_VAR
VAR_INPUT
	Execute		:	BOOL;		(* B *)	(* Start setting position in axis *)
	ScalingFactor	:	LREAL;		(* B *)	(* Position unit [u] / EncoderIncrements *)
	Mode		: 	E_SetScalingFactorMode;	(* E *)
	Options		:	ST_SetEncoderScalingOptions;	(* V *)	(* Beckhoff proprietary input *)
END_VAR
VAR_OUTPUT
	Done		:	BOOL;		(* B *)	(* Position has new value *)
	Busy		:	BOOL;		(* E *)	(* Shows that the Function Block is not finished *)
	Error		:	BOOL;		(* B *)	(* Signals that an error has occurred within the Function Block *)
	ErrorID		:	UDINT;		(* E *)	(* Error identification *)
END_VAR
(*
	Note:
	RELATIVE means that the actual position of the axis is adjusted to the 
	new scaling factor value in a way that no position jump will occur.
	ABSOLUTE means that the scaling factor will be set without any 
	internal position offsets. In this case the actual position value of the 
	axis will jump instantaneously.
	When changing the scaling factor on the fly, RELATIVE mode is 
	supposed to be preferred.
*)
VAR
	ADSbusy	: 	BOOL;
	stSetEncoderSaclingFactor	:	_ST_TcNC_SetEncoderSaclingFactor;
	iState		:	_E_TcMC_STATES := STATE_INITIALIZATION;
	fbAdsWrite	:	ADSWRITE;
END_VAR
{library private}
VAR
	fbOnTrigger	:	R_TRIG;
END_VAR
fbOnTrigger(CLK:= Execute);

CASE iState OF
STATE_INITIALIZATION:
	Busy := FALSE;
	IF NOT Execute THEN
		Done := FALSE;
		Error := FALSE;			(* reset at falling edge of Execute *)
		ErrorID := 0;
	END_IF
	IF fbOnTrigger.Q THEN
		Busy := TRUE;
		(* initialize output values *)
		Done := FALSE;
		Error := FALSE;
		ErrorID := 0;
		fbAdsWrite(WRITE := FALSE);

		(* fill structure*)
		stSetEncoderSaclingFactor.fEncoderScalingFactor := ScalingFactor;
		stSetEncoderSaclingFactor.nEncoderScalingFactorType := Mode;
		stSetEncoderSaclingFactor.nCtrlWord.1 := SEL( Options.SelectEncoderIndex, FALSE, TRUE ); 	(* set bit 1 to explicitly select an encoder / control loop - KSt 2009-04-09 *)

		IF Options.SelectEncoderIndex THEN (* KSt 2009-04-09 *)
			(* select the user defined encoder/control loop explicitly *)
			fbAdsWrite.IDXOFFS:= TcMcGlobal.Axis.Functions.IDXOFFS.SETENCODERSCALING + Options.EncoderIndex * 16#00100000;
		ELSE
			(* select the encoder / control loop that is defined by the AXIS_REF interface
				0  	=  select active encoder / control loop		- used when standard AXIS_REF interface is used
				1..n 	=  explicit encoder / control loop selection 	- used when dedicated encoder AXIS_REF interface is used 		*)
			fbAdsWrite.IDXOFFS:= TcMcGlobal.Axis.Functions.IDXOFFS.SETENCODERSCALING + Axis.NcToPlc.ControlLoopIndex * 16#00100000;
		END_IF

		fbAdsWrite(	NETID:= TcMcGlobal.NCNETID_TCMC,
					PORT:= AMSPORT_R0_NCSAF,
					IDXGRP:=TcMcGlobal.Axis.Functions.IDXGRP+Axis.NcToPlc.AxisId,
(*					IDXOFFS:= TcMcGlobal.Axis.Functions.IDXOFFS.SETENCODERSCALING + Options.EncoderIndex * 16#100000,*) (* KSt 2009-04-09 - see selection above *)
					LEN:= SIZEOF(stSetEncoderSaclingFactor),
					SRCADDR:= ADR(stSetEncoderSaclingFactor),
					WRITE:= TRUE,
					TMOUT:= TcMcGlobal.tADSTimeOut);
		iState := STATE_ORDER;
	END_IF;

STATE_ORDER:
	fbAdsWrite();
	IF NOT fbAdsWrite.Busy THEN
		IF fbAdsWrite.Err THEN
			ErrorID := fbAdsWrite.ErrId;
			Error := TRUE;
		ELSE
			Done := TRUE;
		END_IF;
		fbAdsWrite(WRITE := FALSE);
		iState := STATE_INITIALIZATION;
	END_IF;

ELSE  (* CASE : Unknown program state *)
	Error := TRUE;
	ErrorID := 16#FFFFFFFF;
	iState:= STATE_INITIALIZATION;
END_CASE

ADSbusy := fbAdsWrite.BUSY;

IF iState=STATE_INITIALIZATION THEN
	(* reset Busy immediately  when sequence ends *)
	Busy := FALSE;
END_IF
END_FUNCTION_BLOCK

(* POU MC_SetOverride, ST *)
FUNCTION_BLOCK MC_SetOverride
(*
	This function block sets the values of override for the whole axis, and all 
	functions that are working on that axis. The override parameters act as a factor 
	that is multiplied to the commanded velocity, acceleration, deceleration and jerk 
	of the move function block.
*)
VAR_IN_OUT
	Axis			:	AXIS_REF;
END_VAR
VAR_INPUT
	Enable		:	BOOL;	(* B *)
	VelFactor	:	LREAL	(* B *)	:= 1.0;	(* 1.0 = 100% *)
	AccFactor	:	LREAL	(* E *)	:= 1.0;	(* 1.0 = 100% *)	(* not supported *)
	JerkFactor	:	LREAL 	(* E *)	:= 1.0;	(* 1.0 = 100% *)	(* not supported *)
END_VAR
VAR_OUTPUT
	Enabled		:	BOOL;	(* B *)
	Busy		:	BOOL;	(* E *)
	Error		:	BOOL;	(* B *)
	ErrorID		:	UDINT;	(* E *)
END_VAR
(*
Notes:
   1.	The Input AccFactor acts on positive and negative acceleration (deceleration).
   2.	This Function Block sets the factor. The override factor is valid until a new override is set.
   3.	The default values of the override factor are 1.0.
   4.	The value of the overrides can be between 0.0 and 1.0. 
	The behavior of values > 1.0 is vendor specific. Values < 0.0 are not allowed. 
	The value 0.0 is not allowed for AccFactor and JerkFactor.
   5.	The value 0.0 set to the VelFactor stops the axis without bringing it to the state standstill.
   6.	Override does not act on slave axes. (Axes in the state synchronized motion). 
   7.	The Function Block does not influence the state diagram of the axis.
   8.	VelFactor can be changed at any time and acts directly on the ongoing motion.
   9.	If in Discrete motion, reducing the AccFactor and/or JerkFactor can lead to a 
	position overshoot – a possible cause of damage
 10.	Activating this Function Block on an axis that is under control of MC_PositionProfile, 
	MC_VelocityProfile, or MC_AccelerationProfile, is vendor specific.
*)
VAR
END_VAR
IF Enable THEN
	Busy := TRUE;
	IF VelFactor > 1 OR VelFactor < 0 THEN
		ErrorID := MC_ERROR_PARAMETER_NOT_CORRECT;
		Error := TRUE;
	ELSE
		Axis.PlcToNc.Override := LREAL_TO_UDINT(VelFactor*1000000);
		ErrorID := MC_ERROR_NO_ERROR;
		Error := FALSE;
		Enabled:=TRUE;
	END_IF;
ELSE
	Busy := FALSE;
	Enabled:=FALSE;
	Error := FALSE;			(* reset at falling edge of Execute *)
	ErrorID := 0;
END_IF;
END_FUNCTION_BLOCK

(* POU MC_Stop, ST *)
FUNCTION_BLOCK MC_Stop
(*	This Function Block commands a controlled motion stop and transfers the
	axis to the state 'Stopping'. While the axis is in state Stopping, no other FB 
	can perform any motion on the same axis. After the axis has reached velocity 
	zero, the Done output is set to TRUE immediately. The axis remains in the 
	state 'Stopping' as long as Execute is still TRUE or velocity zero is not yet 
	reached. As soon as 'Done' is set and 'Execute' is FALSE the axis goes to 
	state 'StandStill'.
*)
VAR_IN_OUT
	Axis				:	AXIS_REF;	(* B *)
END_VAR
VAR_INPUT
	Execute			:	BOOL;	(* B *)
	Deceleration		:	LREAL;	(* E *)
	Jerk				:	LREAL;	(* E *)
(*	BufferMode		:	MC_BufferMode;*)	(* E *) (* 2008-06-27 KSt - deleted after PlcOpen corrigendum V0.4 *)
	Options			: 	ST_MoveOptions;	(* optional parameters *)
END_VAR
VAR_OUTPUT
	Done			:	BOOL;	(* B *)
	Busy			: 	BOOL;	(* E *)
	Active			: 	BOOL;	(* E *)
	CommandAborted	:	BOOL;	(* E *)
	Error			:	BOOL;	(* B *)
	ErrorID			:	UDINT;	(* E *)
END_VAR
VAR
	LastExecutionResult: 	_ST_FunctionBlockResults;
	ADSbusy		: 	BOOL;
	MoveGeneric		: 	_FB_MoveUniversalGeneric;
	ReleaseLock		: 	ADSWRITE;
	CmdNo			: 	UINT;
	AxisMotionCommandsLocked		: 	BOOL;
	iState			: 	_E_TcMC_STATES := STATE_INITIALIZATION;
END_VAR
{library private}
VAR
	fbOnTrigger		: 	R_TRIG;
	CounterMotionCommandsLocked: INT;
END_VAR
fbOnTrigger(CLK:= Execute);

CASE iState OF
STATE_INITIALIZATION:	(* *)
	Busy := FALSE;
	Active := FALSE;
	IF NOT Execute THEN
		Done := FALSE;
		CommandAborted := FALSE;
		Error := FALSE;			(* reset at falling edge of Execute *)
		ErrorID := 0;
	END_IF
    	IF fbOnTrigger.Q THEN
		(* initialize output values *)
		Done := FALSE;
		Busy := TRUE;
		Active := FALSE;
		CommandAborted := FALSE;
		Error := FALSE;
		ErrorID := 0;
		ReleaseLock.WRITE:=FALSE;
		iState := STATE_ORDER;
	END_IF

STATE_ORDER :
	(* wait until stop is getting active or axis has stopped for a reason *)
	IF 	MoveGeneric.Active OR
		NOT F_AxisHasJob(Axis.NcToPlc.StateDWord)
		THEN
		Active := TRUE;
		ActStop;
		IF NOT ReleaseLock.BUSY THEN (* may be busy after fast stop retrigger *)
			ReleaseLock.WRITE:=FALSE;
			CounterMotionCommandsLocked := 0;
			iState := STATE_RUNNING;
		END_IF
	ELSIF MoveGeneric.Error OR MoveGeneric.CommandAborted THEN	(* ELSIF added 2009-11-09 KSt *)
		Error := MoveGeneric.Error;
		ErrorID := MoveGeneric.ErrorID;
		CommandAborted := MoveGeneric.CommandAborted;
		IF F_AxisHasJob(Axis.NcToPlc.StateDWord) AND NOT F_AxisMotionCommandsLocked(Axis.NcToPlc.StateDWord) THEN
			iState := STATE_INITIALIZATION; (* command not accepted *)
		ELSIF Execute THEN
			iState := STATE_MOTIONCOMMANDSLOCKED;	(* wait to release after Execute is FALSE *)
		ELSE
			ReleaseLock.WRITE := TRUE;	(* release axis if Execute is already FALSE *)
			iState := STATE_WAITING;
		END_IF
	END_IF

STATE_RUNNING:  (* wait until axis stands still and Execute is FALSE *)
	(* axis is stopping during this state *)
	IF 	NOT MoveGeneric.Busy OR					(* successfully stopped *)
		NOT F_AxisHasJob(Axis.NcToPlc.StateDWord)	(* or in standstill for any other reason *)
		THEN
		Error := MoveGeneric.Error;		(* 2008-11-26 KSt *)
		ErrorID := MoveGeneric.ErrorID;	(* 2008-11-26 KSt *)
		CommandAborted := MoveGeneric.CommandAborted;	(* KSt 2009-04-15 *)
		Done := NOT Error AND NOT CommandAborted;	(* KSt 2009-04-15 *)
		IF Execute THEN
			iState := STATE_MOTIONCOMMANDSLOCKED;
		ELSE
			ReleaseLock.WRITE := TRUE;	(* release axis if Execute is already FALSE *)
			iState := STATE_WAITING;
		END_IF
	END_IF

STATE_MOTIONCOMMANDSLOCKED : 	(* axis is in standstill and axis is locked against motion commands during this state *)
	IF NOT Execute THEN	(* reset outputs if Execute is FALSE *)
		Done := FALSE;
		CommandAborted := FALSE;
		Error := FALSE;
		ErrorID := 0;
		ReleaseLock.WRITE:=TRUE;	(* release axis *)
		CounterMotionCommandsLocked := 0;
		iState := STATE_WAITING;
	END_IF

STATE_WAITING : (* release axis and wait until axis is released *)
	IF NOT Execute THEN	(* reset outputs if Execute is FALSE *)
		Done := FALSE;
		CommandAborted := FALSE;
		Error := FALSE;
		ErrorID := 0;
	END_IF
	ReleaseLock.WRITE:=TRUE;
	ActStop; (* call here - fast reaction required *)
	IF NOT ReleaseLock.BUSY THEN
		IF ReleaseLock.ERR THEN
			Error := TRUE;
			ErrorID := ReleaseLock.ERRID;
			iState := STATE_INITIALIZATION;
		(* ELSIF NOT F_AxisMotionCommandsLocked(Axis.NcToPlc.StateDWord) THEN *) (* NOT deleted 2009-05-11 KSt *)
		ELSIF F_AxisMotionCommandsLocked(Axis.NcToPlc.StateDWord) THEN
			CounterMotionCommandsLocked := CounterMotionCommandsLocked + 1; (* wait for a certain number of cycles before error - 2009-10-06 KSt *)
			IF CounterMotionCommandsLocked > TcMcGlobal.NCTOPLC_FEEDBACK_MAXWAITCYCLES THEN
				Error := TRUE;
				ErrorID := MC_ERROR_BUFFERED_COMMAND_NO_STATE_FEEDBACK; (* lock bit has not been reset *)
				iState := STATE_INITIALIZATION;
			END_IF
		ELSE (* axis released - no error *)
			iState := STATE_INITIALIZATION;
		END_IF
		ReleaseLock.WRITE:=FALSE;
	END_IF

    	IF fbOnTrigger.Q THEN (* KSt 2009-04-15 - Stop retrigger allowed after release even without a "released" feedback*)
		(* initialize output values *)
		Done := FALSE;
		Busy := TRUE;
		Active := FALSE;
		CommandAborted := FALSE;
		Error := FALSE;
		ErrorID := 0;
		ReleaseLock.WRITE:=FALSE;
		iState := STATE_ORDER;	(* retrigger stop command *)
	END_IF

END_CASE

ActStop; (* call function blocks *)

ADSbusy := MoveGeneric.ADSbusy OR ReleaseLock.BUSY;
IF iState=STATE_INITIALIZATION THEN
	(* reset Busy immediately  when sequence ends *)
	Done:=FALSE;
	Busy := FALSE;
	Active := FALSE;
END_IF
END_FUNCTION_BLOCK
ACTION ActStop:
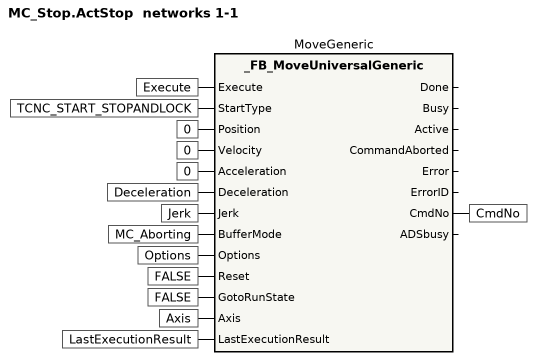
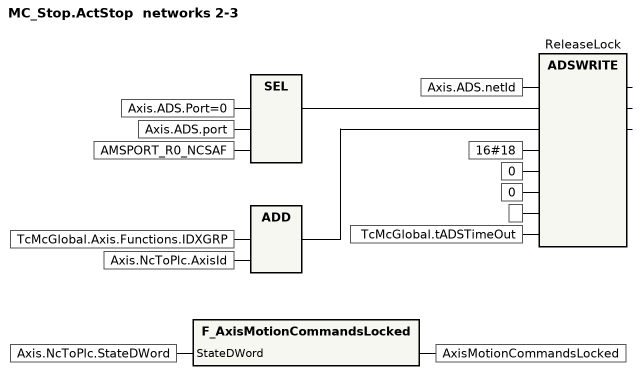
_FBD_ (* Function Block Diagram *)
NETWORK 1
	MoveGeneric:_FB_MoveUniversalGeneric(Execute: Execute, StartType: TCNC_START_STOPANDLOCK, Position: 0, Velocity: 0, Acceleration: 0, Deceleration: Deceleration, Jerk: Jerk, BufferMode: MC_Aborting, Options: Options, Reset: FALSE, GotoRunState: FALSE, Axis: Axis, LastExecutionResult: LastExecutionResult, CmdNo => CmdNo)
NETWORK 2 (* Release locked axis after it has been locked by the MC_Stop command *)
	ReleaseLock:ADSWRITE(Axis.ADS.netId, SEL(Axis.ADS.Port=0, Axis.ADS.port, AMSPORT_R0_NCSAF), ADD(TcMcGlobal.Axis.Functions.IDXGRP, Axis.NcToPlc.AxisId), 16#18, 0, 0, ,  TcMcGlobal.tADSTimeOut)
NETWORK 3
	F_AxisMotionCommandsLocked(StateDWord: Axis.NcToPlc.StateDWord) => AxisMotionCommandsLocked
_END_FBD_
(* the same logic as Structured Text *)
(* Network 1 *)
MoveGeneric(Execute := Execute, StartType := TCNC_START_STOPANDLOCK, Position := 0, Velocity := 0, Acceleration := 0, Deceleration := Deceleration, Jerk := Jerk, BufferMode := MC_Aborting, Options := Options, Reset := FALSE, GotoRunState := FALSE, Axis := Axis, LastExecutionResult := LastExecutionResult);
CmdNo := MoveGeneric.CmdNo;
(* Network 2: see the listing above *)
(* Network 3 *)
AxisMotionCommandsLocked := F_AxisMotionCommandsLocked(StateDWord := Axis.NcToPlc.StateDWord);
END_ACTION

(* POU MC_TouchProbe, ST *)
FUNCTION_BLOCK MC_TouchProbe
(*	The function block is used to record an axis position at a trigger event *)
VAR_IN_OUT
	Axis				:	AXIS_REF; 		(* B *)	(* Identifies the axis which position should be recorded at a defined event at the trigger input *)
	TriggerInput		: 	TRIGGER_REF; 	(* B *)	(* Reference to the trigger signal source. *)
END_VAR
VAR_INPUT
	Execute			:	BOOL;	(* B *)	(* Starts touch probe recording *)
	WindowOnly		: 	BOOL;	(* E *)	(* Enables the monitoring window *)
	FirstPosition		: 	LREAL;	(* E *)	(* Beginning of the monitoring window *)
	LastPosition		: 	LREAL;	(* E *)	(* Ending of the monitoring window *)
END_VAR
VAR_OUTPUT
	Done			:	BOOL;	(* B *)	(* move completed *)
	Busy			: 	BOOL;	(* E *)	(* function block is currently Busy *)
	CommandAborted	: 	BOOL;	(* E *)
	Error			:	BOOL;	(* B *)	(* Signals that error has occurred within Function Block *)
	ErrorID			:	UDINT;	(* E *)	(* Error identification *)
	RecordedPosition:	LREAL;	(* B *)	(* Position where trigger event occurred *)
END_VAR
VAR
	ADSbusy: BOOL;
	iState			: 	_E_TcMC_STATES := STATE_INITIALIZATION;
	TouchProbeValid	: 	ARRAY[1..4] OF UDINT;	(* valid state of probes 1..4 *)
	TouchProbeActive: 	ARRAY[1..4] OF UDINT;	(* activation state of probes 1..4 *)
	TouchProbeValue : 	ARRAY[1..4] OF LREAL;	(* last recorded value of probes 1..4 *)
	TouchProbeModuloValue : 	ARRAY[1..4] OF LREAL;	(* last recorded modulo value of probes 1..4 *)
	TouchProbeInactiveCounter: 	ARRAY[1..4] OF INT;	(* number of cycles where the probes 1..4 where inactive (activation monitoring) *)
END_VAR
{library private}
VAR CONSTANT
	OLDADSINTERFACE : BOOL := TRUE; (* temporary flag to test old and new NC ADS touch probe interface *)
END_VAR
VAR
	fbADSwrite		: 	ADSWRITE;
	fbAdsReadValid	: 	ADSREAD;
	fbAdsReadValue	: 	ADSREAD;
	fbAdsReadState	: 	ADSREAD;
	fbAdsReadModulo: 	ADSREAD;
	TimerAdsReadState: 	TON;
	RtrigPlcEvent		: 	R_TRIG;
	FtrigPlcEvent		: 	F_TRIG;
	fbOnTrigger		: 	R_TRIG;
	LatchID			: 	UDINT;
	Restart			: 	BOOL;	(* restart probe sequence when the trigger was outside the defined window *)
	InWindow		: 	BOOL;	(* probe value is inside the defined window *)
	ModuloFactor		: 	LREAL;	(* axis' modulo factor read from the NC *)
	InitDone			: 	BOOL;	(* initialization on start-up finished *)
	IndexOffset		: 	WORD;
	i: INT;
END_VAR
fbOnTrigger(CLK:= Execute);

CASE iState OF
	STATE_INITIALIZATION :
		Busy := FALSE;
		IF NOT Execute THEN
			Done := FALSE;
			Error := FALSE;			(* reset at falling edge of Execute *)
			ErrorID := 0;
		END_IF

		ActTouchProbeStartupInit;	(* will return InitDone *)

		IF fbOnTrigger.Q THEN
			Restart := TRUE;
		END_IF

		IF Restart THEN
			(* check initialization *)
			Busy := fbAdsReadModulo.BUSY;
			Error := fbAdsReadModulo.ERR;
			ErrorID := fbAdsReadModulo.ERRID;
			IF NOT Busy AND NOT InitDone THEN
				(* initialization error *)
				fbAdsReadModulo(READ:=FALSE);	(* initialize again during next cycle *)
				Restart := FALSE;	(* error *)
			ELSIF InitDone THEN;
				Busy := TRUE;
				IF NOT fbADSwrite.BUSY THEN
					(* initialization *)
					Done := FALSE;
					Error := FALSE;
					ErrorID := 0;
					CommandAborted := FALSE;
					RecordedPosition := 0;
					fbADSwrite(WRITE:=FALSE); (* reset *)
					fbAdsReadValid(READ:=FALSE);
					fbAdsReadValue(READ:=FALSE);
					fbAdsReadState(READ:=FALSE);
					TimerAdsReadState(IN:=FALSE);
					RtrigPlcEvent(CLK:=TriggerInput.PlcEvent);
					FtrigPlcEvent(CLK:=TriggerInput.PlcEvent);
					Restart := FALSE;
					FOR i := 1 TO 4 DO
						TouchProbeInactiveCounter[i] := 0;
					END_FOR
				END_IF

				CASE TriggerInput.Edge OF
					RisingEdge :
						IndexOffset := 16#201;
					FallingEdge:
						IndexOffset := 16#202;
				ELSE (* case *)
					Error := TRUE;
					ErrorID := MC_ERROR_INVALID_TOUCH_PROBE;
				END_CASE

				IF TriggerInput.EncoderID > 255 THEN
					Error := TRUE;
					ErrorID := MC_ERROR_INVALID_TOUCH_PROBE;
				END_IF

				IF NOT Error THEN
					CASE TriggerInput.TouchProbe OF
						TouchProbe1,
						TouchProbe2,
						TouchProbe3,
						TouchProbe4:
							(* activate latch *)
							ActTouchProbeActivate;
							iState := STATE_ORDER;

						PlcEvent:
							(* no action necessary here *);
							TriggerInput.ProbeState := TouchProbeActivated;
							iState := STATE_WAITING;
					ELSE
						Error := TRUE;
						ErrorID := MC_ERROR_INVALID_TOUCH_PROBE;
					END_CASE
				END_IF
			END_IF
		END_IF

	STATE_ORDER :	(* wait until probe is activated *)
		ActTouchProbeActivate;

	STATE_WAITING : (* wait until touch probe was trigerred *)
		CASE TriggerInput.TouchProbe OF (* type of touch probe *)
			TouchProbe1,
			TouchProbe2,
			TouchProbe3,
			TouchProbe4:
				ActTouchProbeMonitorLatchValid;
				IF iState=STATE_WAITING THEN (* still not triggered *)
					ActTouchProbeMonitorActivity;
				END_IF

			(* CASE PlcEvent *)
			PlcEvent : (* touch proble will be triggered through a PLC signal (TriggerInput.PlcEvent) *)
				ActTouchProbeMonitorPlcEvent;
		END_CASE (* type of touch probe *)

		IF NOT Done AND (TriggerInput.ProbeState = TouchProbeAborted) THEN
			(* function block has been aborted by an external MC_AbortTrigger *)
			CommandAborted := TRUE;
			iState := STATE_INITIALIZATION;
		END_IF

		IF iState<> STATE_WAITING THEN
			(* leave the waiting state now *)
			TriggerInput.ProbeState := TouchProbeInactive;
			fbAdsReadModulo(READ:=FALSE);	(* initialize again during next cycle *)
		END_IF
END_CASE

ADSbusy := fbAdsWrite.BUSY OR fbAdsReadValid.BUSY OR fbAdsReadValue.BUSY OR fbAdsReadState.BUSY OR fbAdsReadModulo.BUSY;
IF iState=STATE_INITIALIZATION AND NOT Restart THEN
	(* reset Busy immediately  when sequence ends *)
	Busy := FALSE;
END_IF
END_FUNCTION_BLOCK
ACTION ActTouchProbeActivate:
(* start the touch probe sequence *)

LatchID := TriggerInput.TouchProbe;
TriggerInput.ProbeState := TouchProbeActivated;

fbADSwrite(	NETID:= TcMcGlobal.NCNETID_TCMC,
			PORT:=AMSPORT_R0_NCSAF ,
			IDXGRP:=16#5200+TriggerInput.EncoderID ,
			IDXOFFS:=IndexOffset,
			LEN:=SEL(OLDADSINTERFACE, SIZEOF(LatchID), 0) ,
			SRCADDR:=ADR(LatchID),
			WRITE:=TRUE ,
			TMOUT:=TcMcGlobal.tADSTimeOut);

IF NOT fbADSwrite.BUSY THEN
	IF fbADSwrite.ERR THEN
		Error := fbADSwrite.ERR;
		ErrorID := fbADSwrite.ERRID;
	END_IF
	IF NOT Error AND TriggerInput.ProbeState = TouchProbeAborted THEN
		(* Synchronization error between MC_TouchProbe and MC_AbortTrigger *)
		Error := TRUE;
		ErrorID := MC_ERROR_TOUCH_PROBE_DEACTIVATED;
	END_IF
	TriggerInput.ProbeState := SEL( Error, TouchProbeActivated, TouchProbeInactive );
	iState := SEL( Error, STATE_WAITING, STATE_INITIALIZATION);
END_IF
END_ACTION
ACTION ActTouchProbeMonitorActivity:
(* check if latch is still active *)
TimerAdsReadState(IN := NOT TimerAdsReadState.q , PT:=T#1s);
IF TimerAdsReadState.q OR fbAdsReadState.BUSY THEN
	fbAdsReadState(	NETID:= TcMcGlobal.NCNETID_TCMC,
				PORT:=AMSPORT_R0_NCSAF ,
				IDXGRP:=16#5100+TriggerInput.EncoderID ,
				IDXOFFS:= 16#201,
				LEN:=SEL(OLDADSINTERFACE, SIZEOF(TouchProbeActive), 2),
				DESTADDR:=ADR(TouchProbeActive) ,
				READ:=TRUE ,
				TMOUT:=TcMcGlobal.tADSTimeOut );
	IF NOT fbAdsReadState.BUSY THEN
		IF fbAdsReadState.ERR THEN
			Error := TRUE;
			ErrorID := fbAdsReadState.ERRID;
		ELSE
			IF TouchProbeActive[TriggerInput.TouchProbe]<>1 THEN
				TouchProbeInactiveCounter[TriggerInput.TouchProbe] := TouchProbeInactiveCounter[TriggerInput.TouchProbe] + 1;
				IF TouchProbeInactiveCounter[TriggerInput.TouchProbe] > 1 THEN
					(* error condition when the probing sequence is inactive more than once *)
					Error := TRUE;
					ErrorID := MC_ERROR_TOUCH_PROBE_DEACTIVATED;
					CommandAborted := TRUE;
					iState := STATE_INITIALIZATION;
				END_IF
			END_IF
		END_IF
		fbAdsReadState(READ:=FALSE); (* reset *)
	END_IF
END_IF
END_ACTION
ACTION ActTouchProbeMonitorLatchValid:
(* monitor if the touch probe has been triggered *)

IF F_AxisExternalLatchValid(Axis.NcToPlc.StateDWord) THEN
	(* read the status of the latch *)
	fbAdsReadValid(	NETID:= TcMcGlobal.NCNETID_TCMC,
				PORT:=AMSPORT_R0_NCSAF ,
				IDXGRP:=16#5100+TriggerInput.EncoderID ,
				IDXOFFS:= 16#202,
				LEN:=SEL(OLDADSINTERFACE, SIZEOF(TouchProbeValid), 2) ,
				DESTADDR:=ADR(TouchProbeValid) ,
				READ:=TRUE ,
				TMOUT:=TcMcGlobal.tADSTimeOut );
	(* read the latched value *)
	fbAdsReadValue(	NETID:= TcMcGlobal.NCNETID_TCMC,
				PORT:=AMSPORT_R0_NCSAF ,
				IDXGRP:=16#5100+TriggerInput.EncoderID ,
				IDXOFFS:= 16#205,
				LEN:=SEL(OLDADSINTERFACE, SIZEOF(TouchProbeValue), SIZEOF(TouchProbeValue[1])) ,
				DESTADDR:=ADR(TouchProbeValue) ,
				READ:=TRUE ,
				TMOUT:=TcMcGlobal.tADSTimeOut );
	IF NOT fbAdsReadValid.BUSY AND NOT fbAdsReadValue.BUSY THEN
		IF fbAdsReadValid.err THEN
			Error := TRUE;
			ErrorID := fbAdsReadValid.ERRID;
			iState := STATE_INITIALIZATION;
		ELSIF fbAdsReadValue.err THEN
			Error := TRUE;
			ErrorID := fbAdsReadValue.ERRID;
			iState := STATE_INITIALIZATION;
		ELSE (* no error *)
			IF TouchProbeValid[TriggerInput.TouchProbe]=1 THEN
				RecordedPosition:=TouchProbeValue[TriggerInput.TouchProbe];
				Done := TRUE;
				IF TriggerInput.ModuloPositions AND (ModuloFactor<>0) THEN	(* check for  (ModuloFactor=0) - 2007-02-06 KSt *)
					RecordedPosition :=  ((RecordedPosition / ModuloFactor) - TRUNC(RecordedPosition / ModuloFactor)) * ModuloFactor;
					TouchProbeModuloValue[TriggerInput.TouchProbe] := RecordedPosition;
					InWindow := (RecordedPosition>=FirstPosition) AND (RecordedPosition<=LastPosition);
				ELSE
					InWindow := (RecordedPosition>=FirstPosition) AND (RecordedPosition<=LastPosition);
				END_IF
				IF WindowOnly AND NOT InWindow THEN
					RecordedPosition:=0;
					Done := FALSE;
					Restart := TRUE; (* ignore this event, latch next one *)
				END_IF
				iState := STATE_INITIALIZATION;
			ELSE
				fbAdsReadValid(READ:=FALSE);
				fbAdsReadValue(READ:=FALSE);
			END_IF
		END_IF
	END_IF
END_IF
END_ACTION
ACTION ActTouchProbeMonitorPlcEvent:
(* touch probe sequence for simple PLC inputs *)
(* monitor PLC input trigger *)

RtrigPlcEvent(CLK:=TriggerInput.PlcEvent);
FtrigPlcEvent(CLK:=TriggerInput.PlcEvent);
IF ((TriggerInput.Edge=RisingEdge) AND RtrigPlcEvent.Q) OR
   ((TriggerInput.Edge=FallingEdge) AND FtrigPlcEvent.Q) THEN
	RecordedPosition:=Axis.NcToPlc.ActPos; 	(* 2007-02-06 KSt *)
	IF TriggerInput.ModuloPositions AND (ModuloFactor<>0) THEN	(* check for  (ModuloFactor=0) - 2007-02-06 KSt *)
		RecordedPosition :=  ((RecordedPosition / ModuloFactor) - TRUNC(RecordedPosition / ModuloFactor)) * ModuloFactor;
		InWindow := (RecordedPosition>=FirstPosition) AND (RecordedPosition<=LastPosition);
	ELSE
		InWindow := (RecordedPosition>=FirstPosition) AND (RecordedPosition<=LastPosition);
	END_IF
	IF WindowOnly AND NOT InWindow THEN
		RecordedPosition:=0;	(* 2007-02-06 KSt *)
	ELSE
		Done := TRUE;
		iState := STATE_INITIALIZATION;
	END_IF
END_IF
END_ACTION
ACTION ActTouchProbeStartupInit:
(* initialization on plc start-up *)
(* read the axis' modulo factor *)

IF TriggerInput.ModuloPositions THEN
	IF ModuloFactor = 0 THEN
		InitDone := FALSE; (* 2007-02-06 KSt *)
	END_IF
	fbAdsReadModulo(	NETID:= TcMcGlobal.NCNETID_TCMC,
						PORT:= AMSPORT_R0_NCSAF,
						IDXGRP:= 16#5000+TriggerInput.EncoderID ,
						IDXOFFS:= 16#9,
						LEN:= SIZEOF(ModuloFactor),
						DESTADDR:= ADR(ModuloFactor),
						READ:= TRUE,
						TMOUT:= TcMcGlobal.tADSTimeOut);
	IF NOT fbAdsReadModulo.BUSY THEN
		IF fbAdsReadModulo.ERR OR (ModuloFactor=0) THEN
			fbAdsReadModulo( READ:=FALSE ); 	(* 2007-02-06 KSt *)
			InitDone := FALSE; 	(* init failed - 2007-02-06 KSt *)
			Error := TRUE;
			ErrorID := fbAdsReadModulo.ERRID;
		ELSE
			InitDone := TRUE;
		END_IF
	END_IF
ELSE (* no modulo positions *)
	fbAdsReadModulo( READ:=FALSE );	(* 2007-02-06 KSt *)
	InitDone := TRUE;
END_IF
END_ACTION

(* POU MC_WriteBoolParameter, ST *)
FUNCTION_BLOCK MC_WriteBoolParameter
(*	This Function Block modifies the value of a vendor specific boolean parameter. *)
VAR_IN_OUT
	Axis				:	AXIS_REF;	(* B *)
END_VAR
VAR_INPUT
	Execute			:	BOOL;	(* B *)
	ParameterNumber	:	INT;		(* B *)
	Value			:	BOOL;	(* B *)
END_VAR
VAR_OUTPUT
	Done			:	BOOL;	(* B *)
	Busy			: 	BOOL;	(* E *)
	Error			:	BOOL;	(* B *)
	ErrorID			:	UDINT;	(* E *)
END_VAR
VAR
	ADSbusy		: 	BOOL;
	fbReadWriteParameter: 	_FB_ReadWriteParameter;
END_VAR
{library private}
VAR
	nParatype 		:	_E_ParameterType;
	dwValue 			: 	DWORD;
	lrValue 			: 	LREAL;
	fbTrigger 		: 	R_TRIG;
END_VAR
IF NOT Execute THEN
	Done := FALSE;
	Error := FALSE;			(* reset at falling edge of Execute *)
	ErrorID := 0;
END_IF
fbTrigger(CLK:= Execute);
IF fbTrigger.Q AND NOT Busy THEN
	Busy := TRUE;
	Done := FALSE;
	Error := FALSE;
	ErrorID := MC_ERROR_NO_ERROR;
END_IF;
(* *)
IF Busy THEN
	nParatype := PARAMETERTYPE_BOOL;
	fbReadWriteParameter(Enable:= TRUE, ParameterNumber:= ParameterNumber, Mode:= READWRITEPARAMETERMODE_WRITE,
						ParameterType:=nParatype, Axis:= Axis, ValueLreal:= lrValue, ValueDword := dwValue, ValueBool := Value);
	IF fbReadWriteParameter.Done THEN
		Done := TRUE;
		Busy := FALSE;
		fbReadWriteParameter(Enable:= FALSE, ParameterNumber:= ParameterNumber, Mode:= READWRITEPARAMETERMODE_WRITE,
						ParameterType:= nParatype , Axis:= Axis, ValueLreal:= lrValue, ValueDword := dwValue, ValueBool := Value);
	END_IF;
	IF fbReadWriteParameter.Error THEN
		Busy := FALSE;
		Done := FALSE;
		Error := TRUE;
		ErrorID := fbReadWriteParameter.ErrorID;
		fbReadWriteParameter(Enable:= FALSE, ParameterNumber:= ParameterNumber, Mode:= READWRITEPARAMETERMODE_WRITE,
						ParameterType:= nParatype , Axis:= Axis, ValueLreal:= lrValue, ValueDword := dwValue, ValueBool := Value);
	END_IF;
END_IF;

ADSbusy := fbReadWriteParameter.ADSbusy;
END_FUNCTION_BLOCK

(* POU MC_WriteParameter, ST *)
FUNCTION_BLOCK MC_WriteParameter
(*	This Function Block modifies the value of a vendor specific parameter. *)
VAR_IN_OUT
	Axis				:	AXIS_REF;	(* B *)
END_VAR
VAR_INPUT
	Execute			:	BOOL;		(* B *)
	ParameterNumber	:	INT;			(* B *)
	Value			:	LREAL;		(* B *)
END_VAR
VAR_OUTPUT
	Done			:	BOOL;		(* B *)
	Busy			: 	BOOL;		(* E *)
	Error			:	BOOL;		(* B *)
	ErrorID			:	UDINT;		(* E *)
END_VAR
VAR
	ADSbusy		: 	BOOL;
	fbReadWriteParameter: _FB_ReadWriteParameter;
END_VAR
{library private}
VAR
	nParatype 		:	_E_ParameterType;
	dwValue 			: 	DWORD;
	bValue 			: 	BOOL;
	fbTrigger 		: 	R_TRIG;
END_VAR
IF NOT Execute THEN
	Done := FALSE;
	Error := FALSE;			(* reset at falling edge of Execute *)
	ErrorID := 0;
END_IF
fbTrigger(CLK:= Execute);
IF fbTrigger.Q AND NOT Busy THEN
	Busy := TRUE;
	Done := FALSE;
	Error := FALSE;
	ErrorID := MC_ERROR_NO_ERROR;
END_IF;
(* *)
IF Busy THEN
	nParatype := PARAMETERTYPE_LREAL;
	fbReadWriteParameter(Enable:= TRUE, ParameterNumber:= ParameterNumber, Mode:= READWRITEPARAMETERMODE_WRITE,
						ParameterType:=nParatype, Axis:= Axis, ValueLreal:= Value, ValueDword := dwValue, ValueBool := bValue);
	IF fbReadWriteParameter.Done THEN
		Done := TRUE;
		Busy := FALSE;
		fbReadWriteParameter(Enable:= FALSE, ParameterNumber:= ParameterNumber, Mode:= READWRITEPARAMETERMODE_WRITE,
						ParameterType:= nParatype , Axis:= Axis, ValueLreal:= Value, ValueDword := dwValue, ValueBool := bValue);
	END_IF;
	IF fbReadWriteParameter.Error THEN
		Busy := FALSE;
		Done := FALSE;
		Error := TRUE;
		ErrorID := fbReadWriteParameter.ErrorID;
		fbReadWriteParameter(Enable:= FALSE, ParameterNumber:= ParameterNumber, Mode:= READWRITEPARAMETERMODE_WRITE,
						ParameterType:= nParatype , Axis:= Axis, ValueLreal:= Value, ValueDword := dwValue, ValueBool := bValue);
	END_IF;
END_IF;

ADSbusy := fbReadWriteParameter.ADSbusy;
END_FUNCTION_BLOCK
